FUNCTION_BLOCK F_SEL_E_4 (* selection event-based selection) (generic FB) *)
  PACKAGE eclipse4diac::utils::selection;
  {SET_ATTRIBUTE(eclipse4diac::core::GenericClassName, 'GEN_F_SEL_E')}
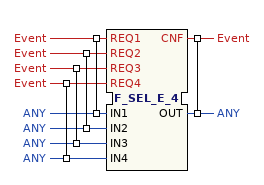
  EVENT_INPUT
    REQ1 WITH IN1;
    REQ2 WITH IN2;
    REQ3 WITH IN3;
    REQ4 WITH IN4;
  END_EVENT
  EVENT_OUTPUT
    CNF WITH OUT; (* Confirmation of Requested Service *)
  END_EVENT
  VAR_INPUT
    IN1 : ANY; (* Selectable input variable *)
    IN2 : ANY; (* Selectable input variable *)
    IN3 : ANY; (* Selectable input variable *)
    IN4 : ANY; (* Selectable input variable *)
  END_VAR
  VAR_OUTPUT
    OUT : ANY; (* Selected input *)
  END_VAR
END_FUNCTION_BLOCK
